VAR_GLOBAL // TIMERS
    ton_p_t: TON;
END_VAR

(* stored: ProductVersion 3.1.0.18, Version 1.1.0.1 *)
